// TIA Portal project "uygulama_1" (V18)

(* hardware
DEVICE "S7-1200 station_1"  S7-1200 Station
   slot 0: "Rack_0"  S7-1200 Rack  Rack  V1.0
   slot 1: "PLC_1"  CPU 1214C DC/DC/DC  6ES7 214-1AG40-0XB0  V4.6
*)

// ===== PLC "PLC_1"  CPU 1214C DC/DC/DC =====

VAR_GLOBAL   // PLC tag table "Default tag table"
   "START" AT %I0.0 : Bool;
   "STOP" AT %I0.1 : Bool;
   "MOTOR1" AT %Q0.0 : Bool;
   "MOTOR2" AT %Q0.1 : Bool;
   "MOTOR3" AT %Q0.2 : Bool;
   "YARDIMCI RÖLE" AT %M0.0 : Bool;
END_VAR

// folder: System blocks/Program resources

DATA_BLOCK "T1"   // DB1
{ S7_Optimized_Access := 'TRUE' }
AUTHOR : Simatic
FAMILY : IEC
NAME : IEC_TMR
VERSION : 1.0
// stored: InstanceOfName IEC_TIMER
"IEC_TIMER"
BEGIN
END_DATA_BLOCK

DATA_BLOCK "T2"   // DB2
{ S7_Optimized_Access := 'TRUE' }
AUTHOR : Simatic
FAMILY : IEC
NAME : IEC_TMR
VERSION : 1.0
// stored: InstanceOfName IEC_TIMER
"IEC_TIMER"
BEGIN
END_DATA_BLOCK

DATA_BLOCK "T3"   // DB3
{ S7_Optimized_Access := 'TRUE' }
AUTHOR : Simatic
FAMILY : IEC
NAME : IEC_TMR
VERSION : 1.0
// stored: InstanceOfName IEC_TIMER
"IEC_TIMER"
BEGIN
END_DATA_BLOCK

DATA_BLOCK "T4"   // DB4
{ S7_Optimized_Access := 'TRUE' }
AUTHOR : Simatic
FAMILY : IEC
NAME : IEC_TMR
VERSION : 1.0
// stored: InstanceOfName IEC_TIMER
"IEC_TIMER"
BEGIN
END_DATA_BLOCK

// folder: (top level)

ORGANIZATION_BLOCK "Main"   // OB1, LAD, ProgramCycle
TITLE = "Main Program Sweep (Cycle)"
{ S7_Optimized_Access := 'TRUE' }
VERSION : 0.1
   VAR_INPUT
      Initial_Call : Bool;   // Initial call of this OB
      Remanence : Bool;   // =True, if remanent data are available
   END_VAR
   VAR_TEMP   // added for the SCL form of the ladder/FBD networks
      _w1 : Bool;
   END_VAR
BEGIN

REGION Network 1
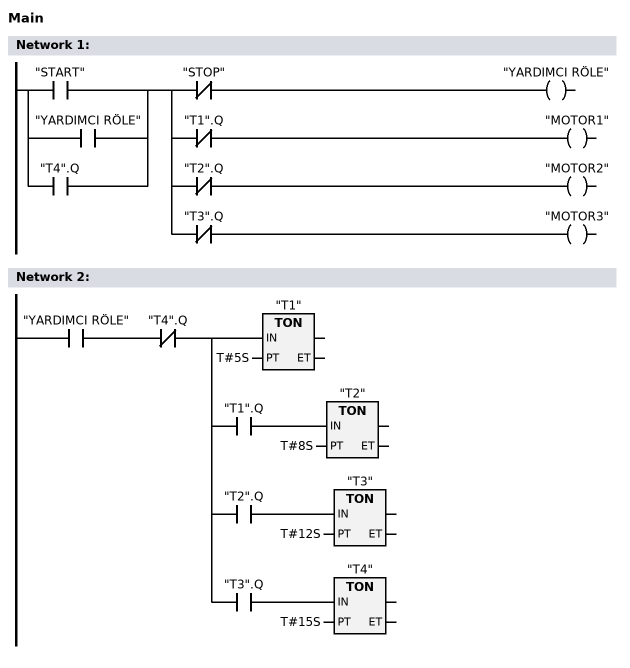
   RUNG wire#powerrail
      Contact( "START" )
      wire#w1
      I_Contact( "STOP" )
      Coil( "YARDIMCI RÖLE" )
   END_RUNG
   RUNG wire#powerrail
      Contact( "YARDIMCI RÖLE" )
   END_RUNG wire#w1
   RUNG wire#powerrail
      Contact( "T4".Q )
   END_RUNG wire#w1
   RUNG wire#w1
      I_Contact( "T1".Q )
      Coil( "MOTOR1" )
   END_RUNG
   RUNG wire#w1
      I_Contact( "T2".Q )
      Coil( "MOTOR2" )
   END_RUNG
   RUNG wire#w1
      I_Contact( "T3".Q )
      Coil( "MOTOR3" )
   END_RUNG
   // the same network as SCL:
   #_w1 := "START" OR "YARDIMCI RÖLE" OR "T4".Q;
   "YARDIMCI RÖLE" := #_w1 AND NOT "STOP";
   "MOTOR1" := #_w1 AND NOT "T1".Q;
   "MOTOR2" := #_w1 AND NOT "T2".Q;
   "MOTOR3" := #_w1 AND NOT "T3".Q;
END_REGION

REGION Network 2
   #_w1 := "YARDIMCI RÖLE" AND NOT "T4".Q;
   "T1".TON(IN := #_w1, PT := T#5S);
   "T2".TON(IN := #_w1 AND "T1".Q, PT := T#8S);
   "T3".TON(IN := #_w1 AND "T2".Q, PT := T#12S);
   "T4".TON(IN := #_w1 AND "T3".Q, PT := T#15S);
END_REGION
END_ORGANIZATION_BLOCK